(* Logix 5000 project; controller Flashing_Light Emulate 5570 rev 30.12; software revision 30.01 *)

TASK MainTask (continuous, watchdog 500 ms) : MainProgram

MODULES
   Local : Emulate 5570 (ICP 2, rev 30.12)
END_MODULES

PROGRAM MainProgram   (* main routine MainRoutine *)
VAR
   Light : BOOL;
   Time1 : TIMER := (PRE := 1000);
   Timer2 : TIMER := (PRE := 1000);
END_VAR

ROUTINE MainRoutine   (* ladder *)
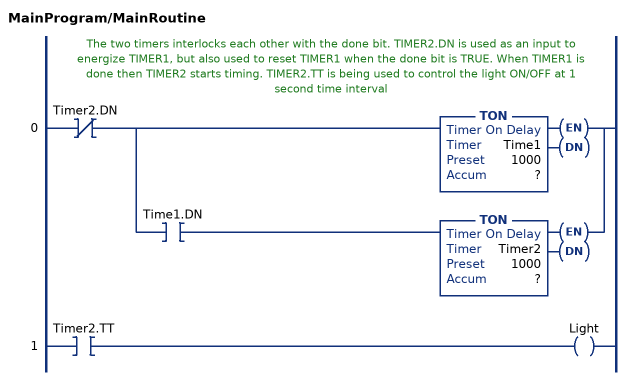
   // The two timers interlocks each other with the done bit. TIMER2.DN is used as an input to energize TIMER1, but also used to reset TIMER1 when the done bit is TRUE. When TIMER1 is done then TIMER2 starts timing. TIMER2.TT is being used to control the light ON/OFF at 1 second time interval
   0: XIO(Timer2.DN)[TON(Time1,?,?) ,XIC(Time1.DN) TON(Timer2,?,?) ];
   1: XIC(Timer2.TT)OTE(Light);
END_ROUTINE
END_PROGRAM
